PROGRAM MAIN_COE_Auswertung
VAR
	COE_Auswertung_0: TwinCAT_Device.Robotino_PLC.COE_Auswertung;
END_VAR

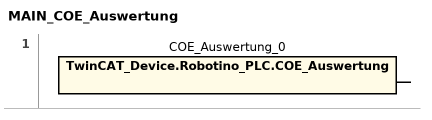
// NETWORK 1
COE_Auswertung_0(); // TwinCAT_Device.Robotino_PLC.COE_Auswertung

END_PROGRAM

(* stored: Version 1.1.0.1, ProductVersion 3.1.4020.12
   POU MAIN_COE_Auswertung: Id {767c06c7-2b13-441a-b1fb-a6f6c3745c0a}, SpecialFunc None *)
